FUNCTION GetPairMasterLength : INT
VAR_INPUT
	pair : REFERENCE TO PositionMaterials;
END_VAR

GetPairMasterLength := MAX(
	GetMaterialLengthFromCode(pair.top),
	GetMaterialLengthFromCode(pair.left),
	GetMaterialLengthFromCode(pair.right),
	GetMaterialLengthFromCode(pair.bottom),
	GetMaterialLengthFromCode(pair.topLeft),
	GetMaterialLengthFromCode(pair.topRight),
	GetMaterialLengthFromCode(pair.bottomLeft),
	GetMaterialLengthFromCode(pair.bottomRight));

END_FUNCTION

(* stored: Version 1.1.0.1, ProductVersion 3.1.4024.11
   POU GetPairMasterLength: Id {dbc8a7af-74ed-4d15-8420-ed1202648c80}, SpecialFunc None *)
